// SIMATIC S7-200 project (STEP 7-Micro/WIN), CPU 222 REL 02.01

ORGANIZATION_BLOCK MAIN:OB1
TITLE=PROGRAM COMMENTS
BEGIN
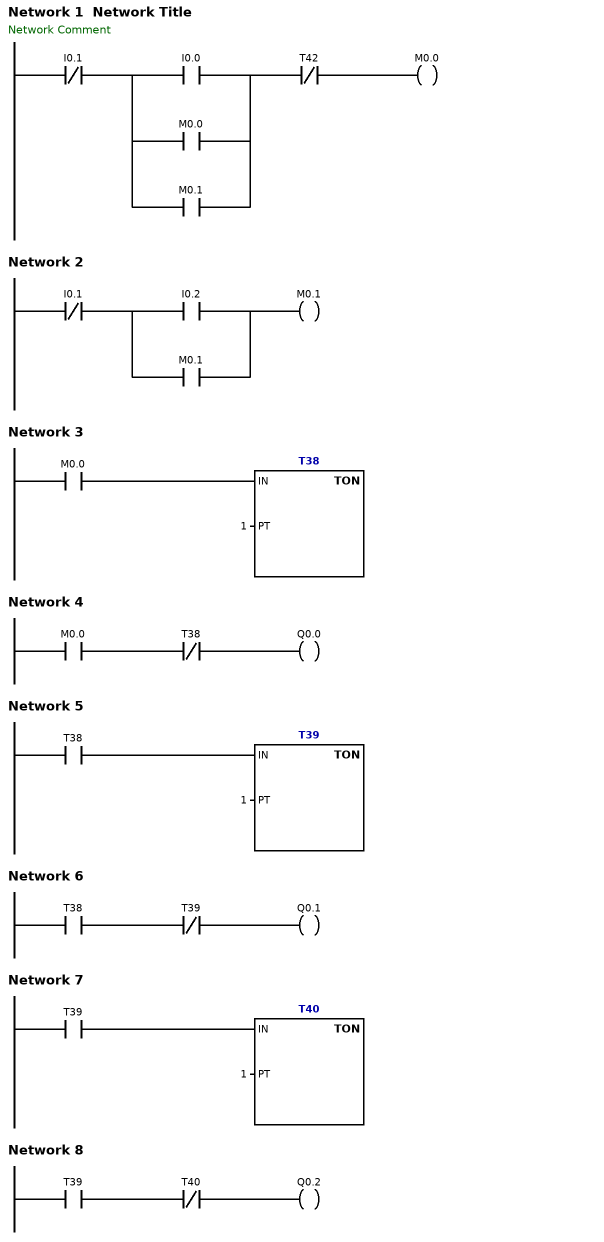
Network 1 // Network Title
// Network Comment
LDN    I0.1
LD     I0.0
O      M0.0
O      M0.1
ALD
AN     T42
=      M0.0
Network 2
LDN    I0.1
LD     I0.2
O      M0.1
ALD
=      M0.1
Network 3
LD     M0.0
TON    T38, 1
Network 4
LD     M0.0
AN     T38
=      Q0.0
Network 5
LD     T38
TON    T39, 1
Network 6
LD     T38
AN     T39
=      Q0.1
Network 7
LD     T39
TON    T40, 1
Network 8
LD     T39
AN     T40
=      Q0.2
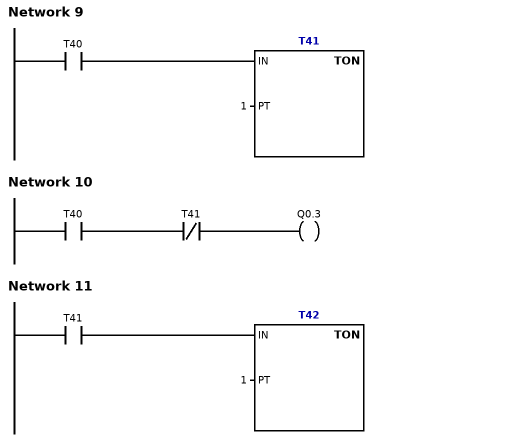
Network 9
LD     T40
TON    T41, 1
Network 10
LD     T40
AN     T41
=      Q0.3
Network 11
LD     T41
TON    T42, 1
END_ORGANIZATION_BLOCK
